Fanuc KAREL source: kt00086.KL

-- PROVISIONAL review KL for V1013-1; original PC SHA256 d00bfcd74314457de15cc859a95ec4de7f122d4b5c253c6449413bdabd2efee6
-- Incomplete behavior may be omitted. Consult companion uncertainty JSON. Do not deploy.
PROGRAM KT00086
%NOLOCKGROUP
VAR
  OUT : REAL
-- UNRESOLVED_DECL Y1 type=002018
-- UNRESOLVED_DECL Y2 type=002018
BEGIN
  -- UNRESOLVED_PC offsets 5-19; opcodes 2E,22,9D,33,B2
  -- UNRESOLVED_PC offsets 24-38; opcodes 2E,22,9D,33,B2
  -- UNRESOLVED_PC offsets 43-57; opcodes 2E,22,9D,33,B2
  -- UNRESOLVED_PC offsets 62-76; opcodes 2E,22,9D,33,B2
  -- UNRESOLVED_PC offsets 81-107; opcodes 22,9D,33,B1,22,9D,33,B1,54,64,23
  -- UNRESOLVED_PC offsets 112-116; opcodes 7F
END KT00086
